// TIA Portal V20 export
VAR_GLOBAL   // PLC tag table "IO_PLC_Centralizer_PLC_Functinal_Test_1"
   In_Functional_Test_Odd AT %I100.0 : "IO_Device_Functinal_Test_Odd";
   Out_Test_Parameters_Odd AT %Q100.0 : "IO_Device_Test_Parameters_Odd";
   Voltage_Read_UInt AT %IW160 : UInt;
END_VAR
